TYPE ST_ClampOutCmd :
STRUCT
    Confirmed : BOOL;
END_STRUCT
END_TYPE

(* stored: Version 1.1.0.1, ProductVersion 3.1.4024.12
   DUT ST_ClampOutCmd: Id {99778224-e186-4d3a-a370-b81169f72d0f} *)
